// TIA Portal project "Simulador" (V15)

(* hardware
DEVICE "S7-1200 station_1"  S7-1200 Station
   slot 0: "Rack_0"  S7-1200 Rack  Rack  V1.0
   slot 1: "PLC_1"  CPU 1214C DC/DC/DC  6ES7 214-1AG40-0XB0  V4.2
*)

// ===== PLC "PLC_1"  CPU 1214C DC/DC/DC =====

VAR_GLOBAL   // PLC tag table "Default tag table"
   ""BtnStop"" AT %I0.1 : Bool;
   ""BtnStart"" AT %I0.2 : Bool;
   ""S2Capacitivo"" AT %I0.3 : Bool;
   ""S1Indutivo"" AT %I0.4 : Bool;
   ""S3Pequeno"" AT %I0.5 : Bool;
   ""S4Medio"" AT %I0.6 : Bool;
   ""S5Grande"" AT %I0.7 : Bool;
   ""SnFinal"" AT %I1.0 : Bool;
   ""Resetar defeito"" AT %I1.3 : Bool;
   ""Motor1"" AT %Q0.1 : Bool;
   ""LampadaSistemaDefeito"" AT %Q2.0 : Bool;
   ""LampadaDefeito"" AT %Q1.0 : Bool;
END_VAR